(* PLC project PLC, Beckhoff Automation GmbH TwinCAT PLC Control 3.5.13.21 *)
(* stored: creationDateTime 2024-02-17T22:42:57.5800916, modificationDateTime 2024-02-17T22:42:57.5800916 *)

TYPE CylResource :
STRUCT
	input: CylInput;
	output: CylOutput;
	config: CylConfig;
	status: CylStatus;
END_STRUCT
END_TYPE
